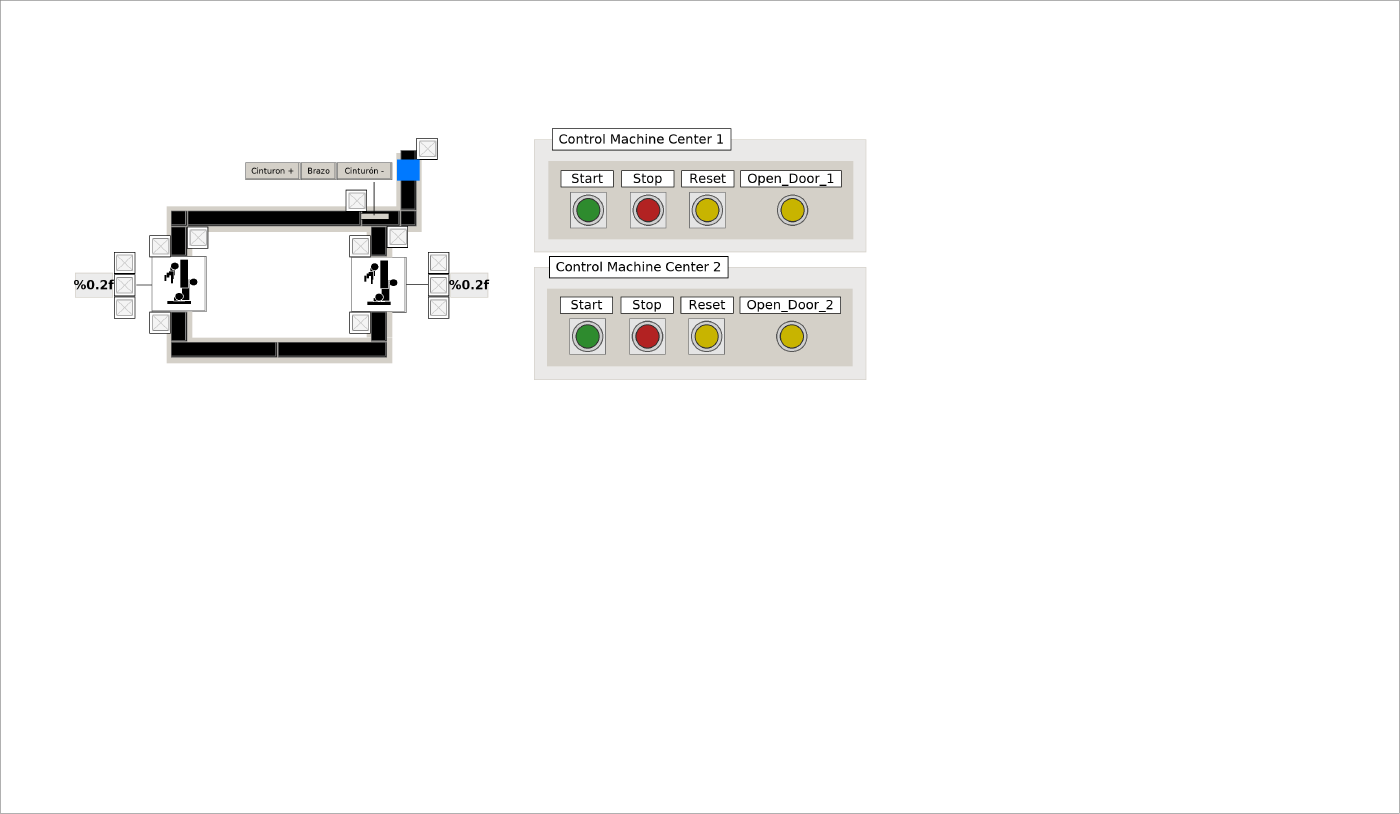
VISUALIZATION Linea_Produccion_Azul_1  // 1940x1128
    Rectangle (1784,668 156x460), angle 90
    Group (487,356 76x81), "2"
        Button (0,0 76x77), pressed state: GVL.Machining_Center_2_Produce_Lids
        RoundedRectangle (35,47 6x34), angle 90
        RoundedRectangle (35,51 6x16), angle 90
        RoundedRectangle (41,31 12x30), angle 47
        Ellipse (32,50 12x11)
        RoundedRectangle (39,4 12x40), angle 130
        Ellipse (52,30 12x11)
        RoundedRectangle (25,11 8x16), angle 24
        Ellipse (26,8 12x11)
        RoundedRectangle (23,20 8x7), angle 24
        RoundedRectangle (27,25 3x6), angle 349
        RoundedRectangle (27,29 2x8), angle 40
        RoundedRectangle (21,23 3x6), angle 259
        RoundedRectangle (18,26 2x8)
    InvisibleInput (82,688 76x76)
    Rectangle (231,286 353x35)
    Rectangle (549,212 35x81)
    Rectangle (231,468 312x35)
    Rectangle (509,321 35x35), angle 90
    Rectangle (230,321 38x35), angle 90
    Group (210,355 76x81), "1"
        Button (0,0 76x77), pressed state: GVL.Machining_Center_1_Produce_Lids
        RoundedRectangle (35,47 6x34), angle 90
        RoundedRectangle (35,51 6x16), angle 90
        RoundedRectangle (41,31 12x30), angle 47
        Ellipse (32,50 12x11)
        RoundedRectangle (39,4 12x40), angle 130
        Ellipse (52,30 12x11)
        RoundedRectangle (25,11 8x16), angle 24
        Ellipse (26,8 12x11)
        RoundedRectangle (23,20 8x7), angle 24
        RoundedRectangle (27,25 3x6), angle 349
        RoundedRectangle (27,29 2x8), angle 40
        RoundedRectangle (21,23 3x6), angle 259
        RoundedRectangle (18,26 2x8)
    Rectangle (509,432 35x35), angle 90
    Rectangle (230,434 38x35), angle 90
    Line (563,394) (593,394)
    Line (210,395) (189,395)
    Rectangle (1784,491 156x460), angle 90
    Rectangle (765,178 248x30), "Control Machine Center 1"
    Rectangle (1793,478 108x422), angle 90
    PushSwitch (790,266 50x50), variable: GVL.Machining_Center_1_Start, behaviour: TOGGLE, style: Switch-PushSwitch-Green
    Rectangle (777,236 73x23), "Start"
    Lamp1 (1073,266 50x50), variable: GVL.Diffuse_Sensor_45, style: Lamp-Lamp1-Yellow
    Rectangle (1026,236 140x23), "Open_Door_1"
    Rectangle (1791,654 107x423), angle 90
    InvisibleInput (1018,652 49x69)
    InvisibleInput (1267,179 49x69)
    InvisibleInput (1090,651 49x69)
    InvisibleInput (1264,0 49x69)
    InvisibleInput (1265,68 49x69)
    Button (555,208 22x83), colour toggle: GVL.Belt_Conveyor_2m_3, pressed state: GVL.Belt_Conveyor_2m_3
        OnMouseClick: toggle GVL.Belt_Conveyor_2m_3
    Group (577,191 29x30), colour toggle: GVL.Diffuse_Sensor_5
        RoundedRectangle (0,0 29x30), colour toggle: GVL.Diffuse_Sensor_4
        Image (4,4 23x22), image: VisuSymbols.Symbols.RSS1
    RoundedRectangle (550,221 31x29)
    Button (555,292 22x21), colour toggle: GVL.Curved_Belt_Conveyor_1_CW, pressed state: GVL.Curved_Belt_Conveyor_1_CW
        OnMouseClick: toggle GVL.Curved_Belt_Conveyor_1_CW
    Button (501,292 53x21), colour toggle: GVL.Belt_Conveyor_2m_4, pressed state: GVL.Belt_Conveyor_2m_4
        OnMouseClick: toggle GVL.Belt_Conveyor_2m_4
    Rectangle (499,295 40x9), angle -45
    Button (260,292 240x21), colour toggle: GVL.Belt_Conveyor_6m_2, pressed state: GVL.Belt_Conveyor_6m_2
        OnMouseClick: toggle GVL.Belt_Conveyor_6m_2
    Button (237,292 22x21), colour toggle: GVL.Curved_Belt_Conveyor_1_CCW, pressed state: GVL.Curved_Belt_Conveyor_1_CCW
        OnMouseClick: toggle GVL.Curved_Belt_Conveyor_1_CCW
    Button (237,314 22x41), colour toggle: GVL.Belt_Conveyor_2m_6, pressed state: GVL.Belt_Conveyor_2m_6
        OnMouseClick: toggle GVL.Belt_Conveyor_2m_6
    Button (514,314 22x41), colour toggle: GVL.Belt_Conveyor_2m_5, pressed state: GVL.Belt_Conveyor_2m_5
        OnMouseClick: toggle GVL.Belt_Conveyor_2m_5
    Button (514,432 22x41), colour toggle: GVL.Belt_Conveyor_2m_14, pressed state: GVL.Belt_Conveyor_2m_14
        OnMouseClick: toggle GVL.Belt_Conveyor_2m_14
    Button (237,432 22x41), colour toggle: GVL.Belt_Conveyor_2m_13, pressed state: GVL.Belt_Conveyor_2m_13
        OnMouseClick: toggle GVL.Belt_Conveyor_2m_13
    Button (237,474 147x21), colour toggle: GVL.Belt_Conveyor_4m_4, pressed state: GVL.Belt_Conveyor_4m_4
        OnMouseClick: toggle GVL.Belt_Conveyor_4m_4
    Button (385,474 151x21), colour toggle: GVL.Belt_Conveyor_4m_5, pressed state: GVL.Belt_Conveyor_4m_5
        OnMouseClick: toggle GVL.Belt_Conveyor_4m_5
    Button (417,225 49x24), "Brazo", colour toggle: GVL.Pivot_Arm_Sorter_2_Turn, pressed state: GVL.Pivot_Arm_Sorter_2_Turn
        OnMouseClick: toggle GVL.Pivot_Arm_Sorter_2_Turn
    Button (340,225 76x24), "Cinturon +", colour toggle: GVL.Pivot_Arm_Sorter_2_Belt_mas, pressed state: GVL.Pivot_Arm_Sorter_2_Belt_mas
        OnMouseClick: toggle GVL.Pivot_Arm_Sorter_2_Belt_mas
    Button (467,225 76x24), "Cinturón -", colour toggle: GVL.Pivot_Arm_Sorter_2_Belt_menos, pressed state: GVL.Pivot_Arm_Sorter_2_Belt_menos
        OnMouseClick: toggle GVL.Pivot_Arm_Sorter_2_Belt_menos
    Line (518,252) (518,298)
    Group (479,263 29x30), colour toggle: GVL.Diffuse_Sensor_6
        RoundedRectangle (0,0 29x30), colour toggle: GVL.Diffuse_Sensor_4
        Image (4,4 23x22), image: VisuSymbols.Symbols.RSS1
    Group (536,313 29x30), colour toggle: GVL.Diffuse_Sensor_7
        RoundedRectangle (0,0 29x30), colour toggle: GVL.Diffuse_Sensor_4
        Image (4,4 23x22), image: VisuSymbols.Symbols.RSS1
    Group (259,314 29x30), colour toggle: GVL.Diffuse_Sensor_8
        RoundedRectangle (0,0 29x30), colour toggle: GVL.Diffuse_Sensor_4
        Image (4,4 23x22), image: VisuSymbols.Symbols.RSS1
    Group (207,432 29x30), colour toggle: GVL.Diffuse_Sensor_17
        RoundedRectangle (0,0 29x30), colour toggle: GVL.Diffuse_Sensor_4
        Image (4,4 23x22), image: VisuSymbols.Symbols.RSS1
    Group (484,432 29x30), colour toggle: GVL.Diffuse_Sensor_18
        RoundedRectangle (0,0 29x30), colour toggle: GVL.Diffuse_Sensor_4
        Image (4,4 23x22), image: VisuSymbols.Symbols.RSS1
    Group (207,326 29x30), colour toggle: GVL.Diffuse_Sensor_15
        RoundedRectangle (0,0 29x30), colour toggle: GVL.Diffuse_Sensor_4
        Image (4,4 23x22), image: VisuSymbols.Symbols.RSS1
    Group (484,326 29x30), colour toggle: GVL.Diffuse_Sensor_16
        RoundedRectangle (0,0 29x30), colour toggle: GVL.Diffuse_Sensor_4
        Image (4,4 23x22), image: VisuSymbols.Symbols.RSS1
    Rectangle (104,378 52x34), "%0.2f", text variable: GVL.Machining_Center_1_Progress
        p4168582468: GVL.Machining_Center_1_Progress
    Group (158,380 29x30), colour toggle: GVL.Machining_Center_1_IsBusy
        RoundedRectangle (0,0 29x30), colour toggle: GVL.Diffuse_Sensor_4
        Image (3,4 23x22), image: VisuSymbols.Symbols.Wheel
    Group (158,349 29x30), colour toggle: GVL.Machining_Center_1_Error
        RoundedRectangle (0,0 29x30), colour toggle: GVL.Diffuse_Sensor_4
        Image (3,4 23x22), image: VisuSymbols.Symbols.Bell
    Group (158,411 29x30), colour toggle: GVL.Machining_Center_1_Opened
        RoundedRectangle (0,0 29x30), colour toggle: GVL.Diffuse_Sensor_4
        Image (3,4 23x22), image: VisuSymbols.Symbols.DoubleArrow3
    Rectangle (624,378 52x34), "%0.2f", text variable: GVL.Machining_Center_1_Progress
        p4168582468: GVL.Machining_Center_1_Progress
    Group (593,380 29x30), colour toggle: GVL.Machining_Center_2_IsBusy
        RoundedRectangle (0,0 29x30), colour toggle: GVL.Diffuse_Sensor_4
        Image (3,4 23x22), image: VisuSymbols.Symbols.Wheel
    Group (593,349 29x30), colour toggle: GVL.Machining_Center_2_Error
        RoundedRectangle (0,0 29x30), colour toggle: GVL.Diffuse_Sensor_4
        Image (3,4 23x22), image: VisuSymbols.Symbols.Bell
    Group (593,411 29x30), colour toggle: GVL.Machining_Center_2_Opened
        RoundedRectangle (0,0 29x30), colour toggle: GVL.Diffuse_Sensor_4
        Image (3,4 23x22), image: VisuSymbols.Symbols.DoubleArrow3
    Rectangle (861,236 73x23), "Stop"
    Rectangle (944,236 73x23), "Reset"
    PushSwitch (873,266 50x50), variable: GVL.Machine_Center_1_Stop, behaviour: TOGGLE, style: Switch-PushSwitch-Red
    PushSwitch (955,266 50x50), variable: GVL.Machine_Center_1_Reset, behaviour: TOGGLE, style: Switch-PushSwitch-Yellow
    PushSwitch (789,441 50x50), variable: GVL.Machining_Center_2_Start, behaviour: TOGGLE, style: Switch-PushSwitch-Green
    Rectangle (776,411 73x23), "Start"
    Lamp1 (1072,441 50x50), variable: GVL.Diffuse_Sensor_46, style: Lamp-Lamp1-Yellow
    Rectangle (1025,411 140x23), "Open_Door_2"
    Rectangle (860,411 73x23), "Stop"
    Rectangle (943,411 73x23), "Reset"
    PushSwitch (872,441 50x50), variable: GVL.Machine_Center_2_Stop, behaviour: TOGGLE, style: Switch-PushSwitch-Red
    PushSwitch (954,441 50x50), variable: GVL.Machine_Center_2_Reset, behaviour: TOGGLE, style: Switch-PushSwitch-Yellow
    Rectangle (761,355 248x30), "Control Machine Center 2"
END_VISUALIZATION

(* stored: Version 1.1.0.1, ProductVersion 3.1.4024.12
   Visu Linea_Produccion_Azul_1: Id {884a9298-ec32-4b73-ba9f-36b715c05151} *)
